// TIA Portal project "TrainingModules" (V15.1)

(* hardware
DEVICE "S71500/ET200MP station_1"  S7-1500 station
   slot 0: "Rail_0"  Rack  6ES7 590-1***0-0AA0
   slot 1: "PLC_1"  CPU 1516-3 PN/DP  6ES7 516-3AN01-0AB0  V2.6
      slot 3: "CPU display_1"  6ES7591-1BA00-0AA0
*)

// ===== PLC "PLC_1"  CPU 1516-3 PN/DP =====

VAR_GLOBAL   // PLC tag table "Default tag table"
   "TT3_Rotated" AT %I12.1 : Bool;   // Input signal the turntable is Rotated TT3
   "TT3_PP_Exit" AT %I12.3 : Bool;   // Input signal a Part Present at the turntable exit TT3
   "CVR2 Contactor FWD" AT %Q10.2 : Bool;   // Activates CVR2 Forward Contactor
END_VAR

VAR_GLOBAL   // PLC tag table "Conveyor Tags"
   "CVR1_Jog_FWD" AT %I10.4 : Bool;   // Manually Jog Conveyor CVR1 Forwards
   "CVR1_Jog_REV" AT %I10.5 : Bool;   // Manually Job Conveyor CVR1 Backwards
   "CVR1 Contactor FWD" AT %Q10.0 : Bool;   // Activates CVR1 Forward Contactor
   "CVR1 Contactor REV" AT %Q10.1 : Bool;   // Activates CVR1 Backward Contactor
   "CVR2 Contactor REV" AT %Q10.3 : Bool;   // Activates CVR2 Backward Contactor
   "CVR3 Contactor FWD" AT %Q10.4 : Bool;   // Activates CVR3 Forward Contactor
   "CVR3 Contactor REV" AT %Q10.5 : Bool;   // Activates CVR3 Backward Contactor
   "CVR2_Jog_FWD" AT %I10.6 : Bool;   // Manually Jog Conveyor CVR2 Forwards
   "CVR2_Jog_REV" AT %I10.7 : Bool;   // Manually Job Conveyor CVR2 Backwards
   "CVR3_Jog_FWD" AT %I11.0 : Bool;   // Manually Jog Conveyor CVR3 Forwards
   "CVR3_Jog_REV" AT %I11.1 : Bool;   // Manually Job Conveyor CVR3 Backwards
   "CVR1_Part_Present" AT %I11.2 : Bool;   // CVR1 Part Present
   "CVR2_Part_Present" AT %I11.3 : Bool;   // CVR2 Part Present
END_VAR

VAR_GLOBAL   // PLC tag table "Turn Table Tags"
   "TT2 Rotate" AT %Q10.6 : Bool;   // Output signals the table to rotate (AUTO Mode) TT2
   "TT2 Rollers FWD" AT %Q10.7 : Bool;   // Output signals the rollers to rotate (AUTO Mode) TT2
   "TT3 Rotate" AT %Q11.0 : Bool;   // Output signals the table to rotate (AUTO Mode) TT3
   "TT3 Rollers FWD" AT %Q11.1 : Bool;   // Output signals the rollers to rotate (AUTO Mode) TT3
   "TT2_Home" AT %I11.4 : Bool;   // Input signal the turntable is Home TT2
   "TT2_Rotated" AT %I11.5 : Bool;   // Input signal the turntable is Rotated TT2
   "TT2_Part_Present" AT %I11.6 : Bool;   // Input signal a Part Present at the turntable entry TT2
   "TT2_PP_Exit" AT %I11.7 : Bool;   // Input signal a Part Present at the turntable exit
   "TT3_Home" AT %I12.0 : Bool;   // Input signal the turntable is Home TT3
   "TT3_Part_Present" AT %I12.2 : Bool;   // Input signal a Part Present at the turntable entry TT3
END_VAR

VAR_GLOBAL   // PLC tag table "Control Panel Tags"
   "AUTO" AT %I10.0 : Bool;   // Auto Switch Enabled
   "AUTO Mode Start" AT %I10.2 : Bool;   // Auto Start PB
   "AUTO Mode Stop" AT %I10.3 : Bool;   // Auto Stop PB
   "Sender" AT %Q12.6 : Bool;   // Parts Sender
   "Receiver" AT %Q12.7 : Bool;   // Parts Receiver
   "Line_Output" AT %QW30 : Word;   // Parts Counter on CVR1
   "MANUAL" AT %I12.4 : Bool;   // Manual Switch Enabled
   "Reset_Counts" AT %I12.6 : Bool;   // Reset Part Counter
   "Conveyor_Estop" AT %I12.7 : Bool;   // Emergency Stop
   "NO MODE" AT %M0.0 : Bool;   // Combines both No Modes into a signal No Modes state
END_VAR

DATA_BLOCK "Conveyor_Line_Status"   // DB450
{ S7_Optimized_Access := 'TRUE' }
VERSION : 0.1
// stored: InstanceOfName GMBlock_Controller
"GMBlock_Controller"
BEGIN
END_DATA_BLOCK

FUNCTION_BLOCK "CVR Logic"   // FB1, LAD
TITLE = Conveyor Logic
{ S7_Optimized_Access := 'TRUE' }
VERSION : 0.1
   VAR_INPUT
      "Auto Switch" : Bool;
      "Auto Mode Start PB" : Bool;
      EStop : Bool;
      "Auto Mode Stop PB" : Bool;
      "Manual Switch" : Bool;
      "Jog FWD PB" : Bool;
      "Part Present" : Bool;
      "Reset Part Count" : Bool;
      "Turn Table Homed" : Bool;
      "Part Loaded" : Bool;
      "No Mode" : Bool;
      "Jog REV PB" : Bool;
   END_VAR
   VAR_OUTPUT
      "Contactor Reverse" : Bool;   // Output signals for rollers to rotate reverse
      "Contactor Forward" : Bool;   // Output signals for rollers to rotate forward
      "Counter Output" : Word;
   END_VAR
   VAR
      "CV Forward Manual" : Bool;
      "CV Forward Auto" : Bool;
   END_VAR
   VAR RETAIN
      "Part Counter" : CTU_INT;
   END_VAR
   VAR
      "Conveyor Started" : Bool;
   END_VAR
   VAR_TEMP   // added for the SCL form of the ladder/FBD networks
      _w1 : Bool;
   END_VAR
BEGIN

REGION Network 1: Conveyor Auto Mode
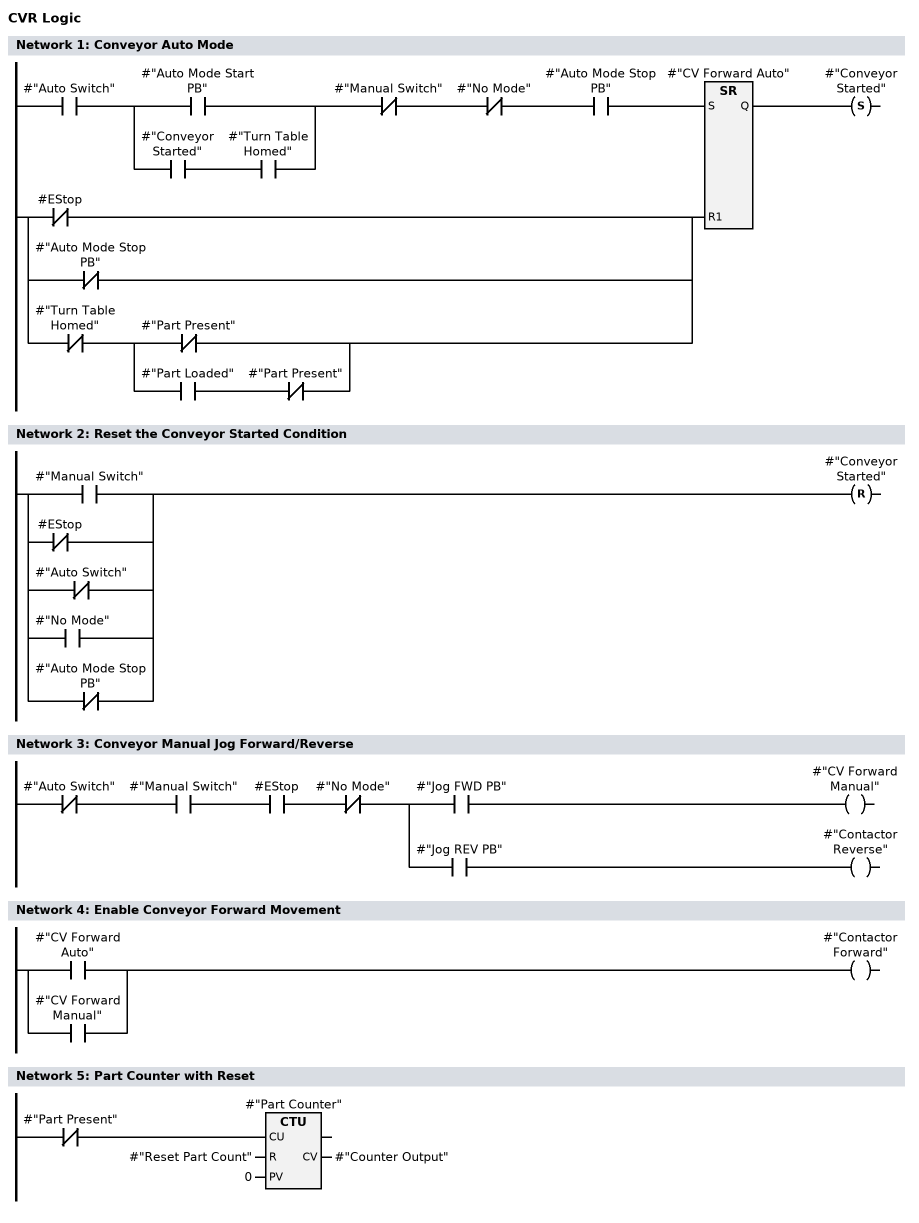
   RUNG wire#powerrail
      Contact( #"Auto Switch" )
      wire#w1
      Contact( #"Auto Mode Start PB" )
      wire#w2
      I_Contact( #"Manual Switch" )
      I_Contact( #"No Mode" )
      Contact( #"Auto Mode Stop PB" )
      S_SR(operand := #"CV Forward Auto", r1 := wire#w4)
      S_Coil( #"Conveyor Started" )
   END_RUNG
   RUNG wire#w1
      Contact( #"Conveyor Started" )
      Contact( #"Turn Table Homed" )
   END_RUNG wire#w2
   RUNG wire#powerrail
      I_Contact( #EStop )
   END_RUNG wire#w4
   RUNG wire#powerrail
      I_Contact( #"Auto Mode Stop PB" )
   END_RUNG wire#w4
   RUNG wire#powerrail
      I_Contact( #"Turn Table Homed" )
      wire#w3
      I_Contact( #"Part Present" )
   END_RUNG wire#w4
   RUNG wire#w3
      Contact( #"Part Loaded" )
      I_Contact( #"Part Present" )
   END_RUNG wire#w4
   // the same network as SCL:
   IF #"Auto Switch" AND (#"Auto Mode Start PB" OR (#"Conveyor Started" AND #"Turn Table Homed")) AND NOT #"Manual Switch" AND NOT #"No Mode" AND #"Auto Mode Stop PB" THEN
       #"CV Forward Auto" := TRUE;   // SR flip-flop
   END_IF;
   IF NOT #EStop OR NOT #"Auto Mode Stop PB" OR (NOT #"Turn Table Homed" AND (NOT #"Part Present" OR (#"Part Loaded" AND NOT #"Part Present"))) THEN
       #"CV Forward Auto" := FALSE;
   END_IF;
   IF #"CV Forward Auto" THEN #"Conveyor Started" := TRUE; END_IF;
END_REGION

REGION Network 2: Reset the Conveyor Started Condition
   RUNG wire#powerrail
      Contact( #"Manual Switch" )
      wire#w1
      R_Coil( #"Conveyor Started" )
   END_RUNG
   RUNG wire#powerrail
      I_Contact( #EStop )
   END_RUNG wire#w1
   RUNG wire#powerrail
      I_Contact( #"Auto Switch" )
   END_RUNG wire#w1
   RUNG wire#powerrail
      Contact( #"No Mode" )
   END_RUNG wire#w1
   RUNG wire#powerrail
      I_Contact( #"Auto Mode Stop PB" )
   END_RUNG wire#w1
   // the same network as SCL:
   IF #"Manual Switch" OR NOT #EStop OR NOT #"Auto Switch" OR #"No Mode" OR NOT #"Auto Mode Stop PB" THEN
       #"Conveyor Started" := FALSE;
   END_IF;
END_REGION

REGION Network 3: Conveyor Manual Jog Forward/Reverse
   RUNG wire#powerrail
      I_Contact( #"Auto Switch" )
      Contact( #"Manual Switch" )
      Contact( #EStop )
      I_Contact( #"No Mode" )
      wire#w1
      Contact( #"Jog FWD PB" )
      Coil( #"CV Forward Manual" )
   END_RUNG
   RUNG wire#w1
      Contact( #"Jog REV PB" )
      Coil( #"Contactor Reverse" )
   END_RUNG
   // the same network as SCL:
   #_w1 := NOT #"Auto Switch" AND #"Manual Switch" AND #EStop AND NOT #"No Mode";
   #"CV Forward Manual" := #_w1 AND #"Jog FWD PB";
   #"Contactor Reverse" := #_w1 AND #"Jog REV PB";
END_REGION

REGION Network 4: Enable Conveyor Forward Movement
   RUNG wire#powerrail
      Contact( #"CV Forward Auto" )
      wire#w1
      Coil( #"Contactor Forward" )
   END_RUNG
   RUNG wire#powerrail
      Contact( #"CV Forward Manual" )
   END_RUNG wire#w1
   // the same network as SCL:
   #"Contactor Forward" := #"CV Forward Auto" OR #"CV Forward Manual";
END_REGION

REGION Network 5: Part Counter with Reset
   #"Part Counter"(CU := NOT #"Part Present", R := #"Reset Part Count", PV := 0, CV => #"Counter Output");   // CTU
END_REGION
END_FUNCTION_BLOCK

FUNCTION_BLOCK "GMBlock_Controller"   // FB2, LAD
TITLE = Conveyor and Turn Table Control Hub
{ S7_Optimized_Access := 'TRUE' }
VERSION : 0.1
   VAR
      CVR1 : "CVR Logic";
      CVR2 : "CVR Logic";
      CVR3 : "CVR Logic";
      TT2 : "TT Logic";
      TT3 : "TT Logic";
   END_VAR
BEGIN

REGION Network 1: Send and Receive Call
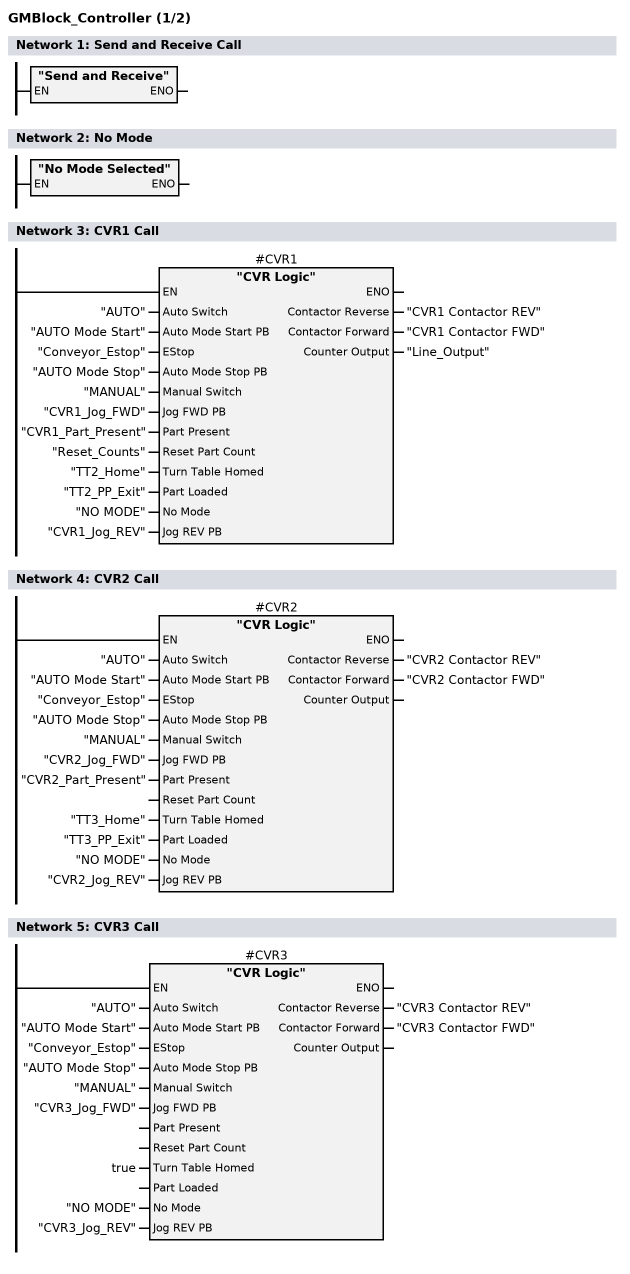
   RUNG wire#powerrail
      "Send and Receive"()
   END_RUNG
   // the same network as SCL:
   "Send and Receive"();
END_REGION

REGION Network 2: No Mode
   RUNG wire#powerrail
      "No Mode Selected"()
   END_RUNG
   // the same network as SCL:
   "No Mode Selected"();
END_REGION

REGION Network 3: CVR1 Call
   RUNG wire#powerrail
      #CVR1("Auto Switch" := "AUTO", "Auto Mode Start PB" := "AUTO Mode Start", EStop := "Conveyor_Estop", "Auto Mode Stop PB" := "AUTO Mode Stop", "Manual Switch" := "MANUAL", "Jog FWD PB" := "CVR1_Jog_FWD", "Part Present" := "CVR1_Part_Present", "Reset Part Count" := "Reset_Counts", "Turn Table Homed" := "TT2_Home", "Part Loaded" := "TT2_PP_Exit", "No Mode" := "NO MODE", "Jog REV PB" := "CVR1_Jog_REV", "Contactor Reverse" => "CVR1 Contactor REV", "Contactor Forward" => "CVR1 Contactor FWD", "Counter Output" => "Line_Output")
   END_RUNG
   // the same network as SCL:
   #CVR1("Auto Switch" := "AUTO",   // "CVR Logic"
         "Auto Mode Start PB" := "AUTO Mode Start",
         EStop := "Conveyor_Estop",
         "Auto Mode Stop PB" := "AUTO Mode Stop",
         "Manual Switch" := "MANUAL",
         "Jog FWD PB" := "CVR1_Jog_FWD",
         "Part Present" := "CVR1_Part_Present",
         "Reset Part Count" := "Reset_Counts",
         "Turn Table Homed" := "TT2_Home",
         "Part Loaded" := "TT2_PP_Exit",
         "No Mode" := "NO MODE",
         "Jog REV PB" := "CVR1_Jog_REV",
         "Contactor Reverse" => "CVR1 Contactor REV",
         "Contactor Forward" => "CVR1 Contactor FWD",
         "Counter Output" => "Line_Output");
END_REGION

REGION Network 4: CVR2 Call
   RUNG wire#powerrail
      #CVR2("Auto Switch" := "AUTO", "Auto Mode Start PB" := "AUTO Mode Start", EStop := "Conveyor_Estop", "Auto Mode Stop PB" := "AUTO Mode Stop", "Manual Switch" := "MANUAL", "Jog FWD PB" := "CVR2_Jog_FWD", "Part Present" := "CVR2_Part_Present", "Reset Part Count" :=, "Turn Table Homed" := "TT3_Home", "Part Loaded" := "TT3_PP_Exit", "No Mode" := "NO MODE", "Jog REV PB" := "CVR2_Jog_REV", "Contactor Reverse" => "CVR2 Contactor REV", "Contactor Forward" => "CVR2 Contactor FWD", "Counter Output" =>)
   END_RUNG
   // the same network as SCL:
   #CVR2("Auto Switch" := "AUTO",   // "CVR Logic"
         "Auto Mode Start PB" := "AUTO Mode Start",
         EStop := "Conveyor_Estop",
         "Auto Mode Stop PB" := "AUTO Mode Stop",
         "Manual Switch" := "MANUAL",
         "Jog FWD PB" := "CVR2_Jog_FWD",
         "Part Present" := "CVR2_Part_Present",
         "Turn Table Homed" := "TT3_Home",
         "Part Loaded" := "TT3_PP_Exit",
         "No Mode" := "NO MODE",
         "Jog REV PB" := "CVR2_Jog_REV",
         "Contactor Reverse" => "CVR2 Contactor REV",
         "Contactor Forward" => "CVR2 Contactor FWD");
END_REGION

REGION Network 5: CVR3 Call
   RUNG wire#powerrail
      #CVR3("Auto Switch" := "AUTO", "Auto Mode Start PB" := "AUTO Mode Start", EStop := "Conveyor_Estop", "Auto Mode Stop PB" := "AUTO Mode Stop", "Manual Switch" := "MANUAL", "Jog FWD PB" := "CVR3_Jog_FWD", "Part Present" :=, "Reset Part Count" :=, "Turn Table Homed" := true, "Part Loaded" :=, "No Mode" := "NO MODE", "Jog REV PB" := "CVR3_Jog_REV", "Contactor Reverse" => "CVR3 Contactor REV", "Contactor Forward" => "CVR3 Contactor FWD", "Counter Output" =>)
   END_RUNG
   // the same network as SCL:
   #CVR3("Auto Switch" := "AUTO",   // "CVR Logic"
         "Auto Mode Start PB" := "AUTO Mode Start",
         EStop := "Conveyor_Estop",
         "Auto Mode Stop PB" := "AUTO Mode Stop",
         "Manual Switch" := "MANUAL",
         "Jog FWD PB" := "CVR3_Jog_FWD",
         "Turn Table Homed" := true,
         "No Mode" := "NO MODE",
         "Jog REV PB" := "CVR3_Jog_REV",
         "Contactor Reverse" => "CVR3 Contactor REV",
         "Contactor Forward" => "CVR3 Contactor FWD");
END_REGION

REGION Network 6: TT2 Call
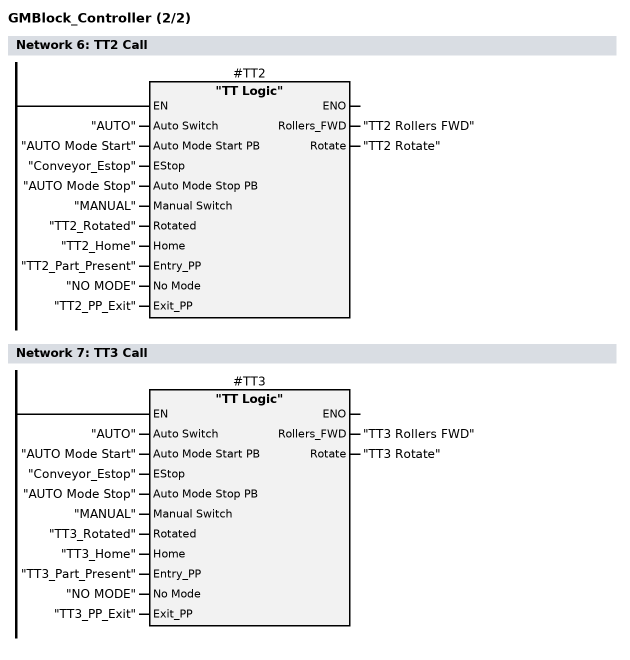
   RUNG wire#powerrail
      #TT2("Auto Switch" := "AUTO", "Auto Mode Start PB" := "AUTO Mode Start", EStop := "Conveyor_Estop", "Auto Mode Stop PB" := "AUTO Mode Stop", "Manual Switch" := "MANUAL", Rotated := "TT2_Rotated", Home := "TT2_Home", Entry_PP := "TT2_Part_Present", "No Mode" := "NO MODE", Exit_PP := "TT2_PP_Exit", Rollers_FWD => "TT2 Rollers FWD", Rotate => "TT2 Rotate")
   END_RUNG
   // the same network as SCL:
   #TT2("Auto Switch" := "AUTO",   // "TT Logic"
        "Auto Mode Start PB" := "AUTO Mode Start",
        EStop := "Conveyor_Estop",
        "Auto Mode Stop PB" := "AUTO Mode Stop",
        "Manual Switch" := "MANUAL",
        Rotated := "TT2_Rotated",
        Home := "TT2_Home",
        Entry_PP := "TT2_Part_Present",
        "No Mode" := "NO MODE",
        Exit_PP := "TT2_PP_Exit",
        Rollers_FWD => "TT2 Rollers FWD",
        Rotate => "TT2 Rotate");
END_REGION

REGION Network 7: TT3 Call
   RUNG wire#powerrail
      #TT3("Auto Switch" := "AUTO", "Auto Mode Start PB" := "AUTO Mode Start", EStop := "Conveyor_Estop", "Auto Mode Stop PB" := "AUTO Mode Stop", "Manual Switch" := "MANUAL", Rotated := "TT3_Rotated", Home := "TT3_Home", Entry_PP := "TT3_Part_Present", "No Mode" := "NO MODE", Exit_PP := "TT3_PP_Exit", Rollers_FWD => "TT3 Rollers FWD", Rotate => "TT3 Rotate")
   END_RUNG
   // the same network as SCL:
   #TT3("Auto Switch" := "AUTO",   // "TT Logic"
        "Auto Mode Start PB" := "AUTO Mode Start",
        EStop := "Conveyor_Estop",
        "Auto Mode Stop PB" := "AUTO Mode Stop",
        "Manual Switch" := "MANUAL",
        Rotated := "TT3_Rotated",
        Home := "TT3_Home",
        Entry_PP := "TT3_Part_Present",
        "No Mode" := "NO MODE",
        Exit_PP := "TT3_PP_Exit",
        Rollers_FWD => "TT3 Rollers FWD",
        Rotate => "TT3 Rotate");
END_REGION
END_FUNCTION_BLOCK

FUNCTION_BLOCK "TT Logic"   // FB3, LAD
{ S7_Optimized_Access := 'TRUE' }
VERSION : 0.1
   VAR_INPUT
      "Auto Switch" : Bool;
      "Auto Mode Start PB" : Bool;
      EStop : Bool;
      "Auto Mode Stop PB" : Bool;
      "Manual Switch" : Bool;
      Rotated : Bool;   // Input signal the turntable is Rotated
      Home : Bool;   // Input signal the turntable is Home
      Entry_PP : Bool;   // Input signal a Part Present at the turntable entry
      "No Mode" : Bool;
      Exit_PP : Bool;   // Input signal a Part Present at the turntable exit
   END_VAR
   VAR_OUTPUT
      Rollers_FWD : Bool;   // Output signals the rollers to rotate (AUTO Mode)
      Rotate : Bool;   // Output signals the table to rotate (AUTO Mode)
   END_VAR
   VAR
      Dropoff_Rollers_FWD : Bool;
      Pickup_Rollers_FWD : Bool;
      "Elapsed Time" : Time;
      "Turn Table Timers" : TP_TIME;
      "Auto Stopped" : Bool;
   END_VAR
BEGIN

REGION Network 1: Enable FWD Rollers on Turn Tables
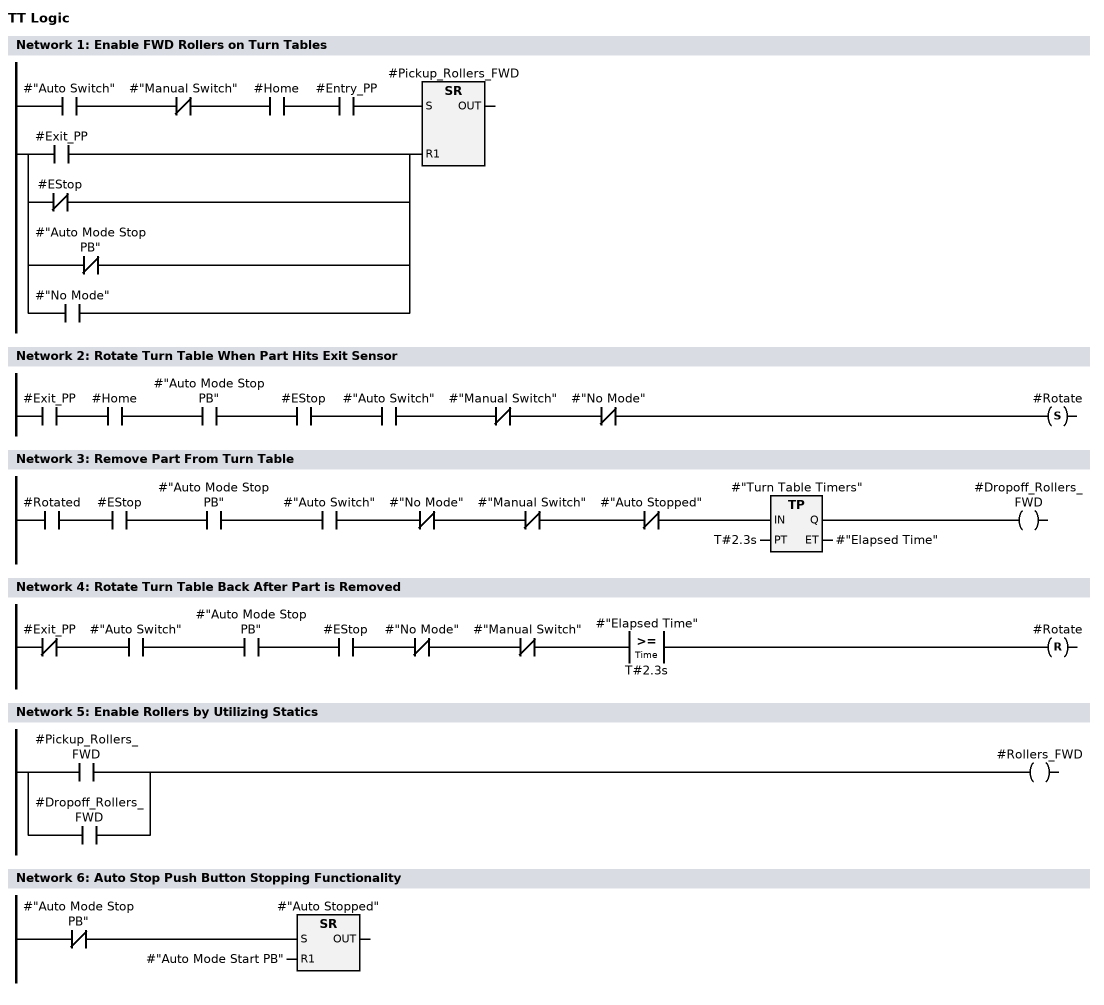
   RUNG wire#powerrail
      Contact( #"Auto Switch" )
      I_Contact( #"Manual Switch" )
      Contact( #Home )
      Contact( #Entry_PP )
      S_SR(operand := #Pickup_Rollers_FWD, r1 := wire#w1)
   END_RUNG
   RUNG wire#powerrail
      Contact( #Exit_PP )
   END_RUNG wire#w1
   RUNG wire#powerrail
      I_Contact( #EStop )
   END_RUNG wire#w1
   RUNG wire#powerrail
      I_Contact( #"Auto Mode Stop PB" )
   END_RUNG wire#w1
   RUNG wire#powerrail
      Contact( #"No Mode" )
   END_RUNG wire#w1
   // the same network as SCL:
   IF #"Auto Switch" AND NOT #"Manual Switch" AND #Home AND #Entry_PP THEN
       #Pickup_Rollers_FWD := TRUE;   // SR flip-flop
   END_IF;
   IF #Exit_PP OR NOT #EStop OR NOT #"Auto Mode Stop PB" OR #"No Mode" THEN
       #Pickup_Rollers_FWD := FALSE;
   END_IF;
END_REGION

REGION Network 2: Rotate Turn Table When Part Hits Exit Sensor
   RUNG wire#powerrail
      Contact( #Exit_PP )
      Contact( #Home )
      Contact( #"Auto Mode Stop PB" )
      Contact( #EStop )
      Contact( #"Auto Switch" )
      I_Contact( #"Manual Switch" )
      I_Contact( #"No Mode" )
      S_Coil( #Rotate )
   END_RUNG
   // the same network as SCL:
   IF #Exit_PP AND #Home AND #"Auto Mode Stop PB" AND #EStop AND #"Auto Switch" AND NOT #"Manual Switch" AND NOT #"No Mode" THEN
       #Rotate := TRUE;
   END_IF;
END_REGION

REGION Network 3: Remove Part From Turn Table
   #"Turn Table Timers"(IN := #Rotated AND #EStop AND #"Auto Mode Stop PB" AND #"Auto Switch" AND NOT #"No Mode" AND NOT #"Manual Switch" AND NOT #"Auto Stopped",   // TP
                        PT := T#2.3s,
                        ET => #"Elapsed Time");
   #Dropoff_Rollers_FWD := #"Turn Table Timers".Q;
END_REGION

REGION Network 4: Rotate Turn Table Back After Part is Removed
   RUNG wire#powerrail
      I_Contact( #Exit_PP )
      Contact( #"Auto Switch" )
      Contact( #"Auto Mode Stop PB" )
      Contact( #EStop )
      I_Contact( #"No Mode" )
      I_Contact( #"Manual Switch" )
      { S7_Templates := "SrcType := Time" } GE_Contact(in1 := #"Elapsed Time", in2 := T#2.3s)
      R_Coil( #Rotate )
   END_RUNG
   // the same network as SCL:
   IF NOT #Exit_PP AND #"Auto Switch" AND #"Auto Mode Stop PB" AND #EStop AND NOT #"No Mode" AND NOT #"Manual Switch" AND (#"Elapsed Time" >= T#2.3s) THEN
       #Rotate := FALSE;
   END_IF;
END_REGION

REGION Network 5: Enable Rollers by Utilizing Statics
   RUNG wire#powerrail
      Contact( #Pickup_Rollers_FWD )
      wire#w1
      Coil( #Rollers_FWD )
   END_RUNG
   RUNG wire#powerrail
      Contact( #Dropoff_Rollers_FWD )
   END_RUNG wire#w1
   // the same network as SCL:
   #Rollers_FWD := #Pickup_Rollers_FWD OR #Dropoff_Rollers_FWD;
END_REGION

REGION Network 6: Auto Stop Push Button Stopping Functionality
   RUNG wire#powerrail
      I_Contact( #"Auto Mode Stop PB" )
      S_SR(operand := #"Auto Stopped", r1 := #"Auto Mode Start PB")
   END_RUNG
   // the same network as SCL:
   IF NOT #"Auto Mode Stop PB" THEN
       #"Auto Stopped" := TRUE;   // SR flip-flop
   END_IF;
   IF #"Auto Mode Start PB" THEN #"Auto Stopped" := FALSE; END_IF;
END_REGION
END_FUNCTION_BLOCK

FUNCTION "Send and Receive" : Void   // FC1, LAD
{ S7_Optimized_Access := 'TRUE' }
VERSION : 0.1
BEGIN

REGION Network 1: Send and Receive Parts in Auto Mode
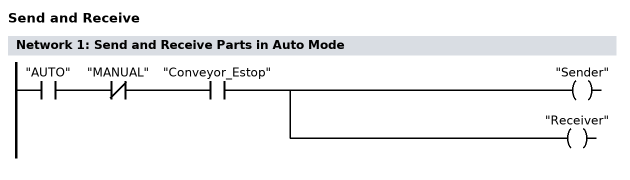
   RUNG wire#powerrail
      Contact( "AUTO" )
      I_Contact( "MANUAL" )
      Contact( "Conveyor_Estop" )
      wire#w1
      Coil( "Sender" )
   END_RUNG
   RUNG wire#w1
      Coil( "Receiver" )
   END_RUNG
   // the same network as SCL:
   "Sender" := "AUTO" AND NOT "MANUAL" AND "Conveyor_Estop";
   "Receiver" := "Sender";
END_REGION
END_FUNCTION

FUNCTION "No Mode Selected" : Void   // FC2, LAD
{ S7_Optimized_Access := 'TRUE' }
VERSION : 0.1
BEGIN

REGION Network 1: Combines both No Modes into a signal No Modes state
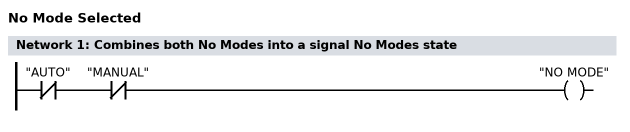
   RUNG wire#powerrail
      I_Contact( "AUTO" )
      I_Contact( "MANUAL" )
      Coil( "NO MODE" )
   END_RUNG
   // the same network as SCL:
   "NO MODE" := NOT "AUTO" AND NOT "MANUAL";
END_REGION
END_FUNCTION

ORGANIZATION_BLOCK "Main"   // OB1, LAD, ProgramCycle
TITLE = "Main Program Sweep (Cycle)"
{ S7_Optimized_Access := 'TRUE' }
VERSION : 0.1
   VAR_INPUT
      Initial_Call : Bool;   // Initial call of this OB
      Remanence : Bool;   // =True, if remanent data are available
   END_VAR
BEGIN

REGION Network 1: GMBlock Controller
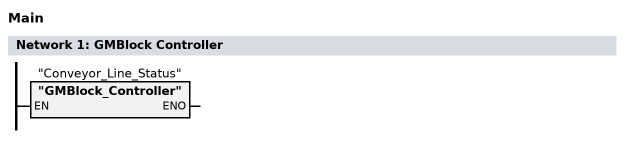
   RUNG wire#powerrail
      "Conveyor_Line_Status"()
   END_RUNG
   // the same network as SCL:
   "Conveyor_Line_Status"();   // "GMBlock_Controller"
END_REGION
END_ORGANIZATION_BLOCK